{attribute 'Tc2GvlVarNames'}
VAR_GLOBAL RETAIN

END_VAR

(* stored: Version 1.1.0.1, ProductVersion 3.1.4022.7
   GVL Setup_Data: Id {283a5430-37f8-4d89-bfd2-38eafe8e246c} *)
